{attribute 'qualified_only'}
VAR_GLOBAL CONSTANT
	NUMBER_OF_JOINTS : INT := 4;
END_VAR

(* stored: Version 1.1.0.1, ProductVersion 3.1.4024.9
   GVL GVL_RobotArm: Id {e11dfeeb-804f-45f2-8083-9d8460acbc0f} *)
